{attribute 'GeneratedUsingTerminal: EL6201-0000-0018'}
{attribute addProperty BoxType "EL6201-0000-0018"}
{attribute addProperty Id "Configuration_okayAT %I*BOOL1Power_FailAT %I*BOOL1Auto_addresing_mode_enabledAT %I*BOOL1Auto_addressing_mode_availableAT %I*BOOL1Protected_mode_activeAT %I*BOOL1Slave_with_address_0_foundAT %I*BOOL1Offline_ReadyAT %I*BOOL1Normal_OperationAT %I*BOOL1ASI_phaseAT %I*BYTE1Power24_Mode_EnabledAT %I*BOOL1Power24_FailAT %I*BOOL1M4_Profile_Support_EnabledAT %I*BOOL1TxPDO_ToggleAT %I*BOOL1"}
{attribute addProperty CRC "664549635"}
{attribute addProperty Size "13"}
TYPE ASI_Status_279C3903 :
STRUCT
	{attribute addProperty Name "Configuration_okay"}
	Configuration_okay AT %I* : BOOL;
	{attribute addProperty Name "Power_Fail"}
	Power_Fail AT %I* : BOOL;
	{attribute addProperty Name "Auto_addresing_mode_enabled"}
	Auto_addresing_mode_enabled AT %I* : BOOL;
	{attribute addProperty Name "Auto_addressing_mode_available"}
	Auto_addressing_mode_available AT %I* : BOOL;
	{attribute addProperty Name "Protected_mode_active"}
	Protected_mode_active AT %I* : BOOL;
	{attribute addProperty Name "Slave_with_address_0_found"}
	Slave_with_address_0_found AT %I* : BOOL;
	{attribute addProperty Name "Offline_Ready"}
	Offline_Ready AT %I* : BOOL;
	{attribute addProperty Name "Normal_Operation"}
	Normal_Operation AT %I* : BOOL;
	{attribute addProperty Name "ASI_phase"}
	ASI_phase AT %I* : BYTE;
	{attribute addProperty Name "Power24_Mode_Enabled"}
	Power24_Mode_Enabled AT %I* : BOOL;
	{attribute addProperty Name "Power24_Fail"}
	Power24_Fail AT %I* : BOOL;
	{attribute addProperty Name "M4_Profile_Support_Enabled"}
	M4_Profile_Support_Enabled AT %I* : BOOL;
	{attribute addProperty Name "TxPDO_Toggle"}
	TxPDO_Toggle AT %I* : BOOL;
END_STRUCT
END_TYPE

(* stored: Version 1.2.0.0, ProductVersion 3.1.4024.9
   DUT ASI_Status_279C3903: Id {7938a123-adff-466c-9529-048286730839} *)
